//Extend the base statusses with project statusses
TYPE HMI_STS_SafetyZone1 EXTENDS HMI_STS_SafetyLogic:
STRUCT
	CrcCodeProject:WORD;		//CRC code safety project
END_STRUCT
END_TYPE

(* stored: Version 1.1.0.1
   DUT HMI_STS_SafetyZone1: Id {50f4144c-cfd0-019f-281a-6ed87517e512} *)
